FUNCTION_BLOCK Gebhardt_Speed
VAR_INPUT
	EN: BOOL;
	ModbusRTU: REFERENCE TO ModbusRTU;
	Address: BYTE := 101;
END_VAR
VAR_OUTPUT
	ENO: BOOL;
	Speed: LREAL;
END_VAR
VAR
	ModbusWord_T_Speed: ModbusReadWord;
END_VAR

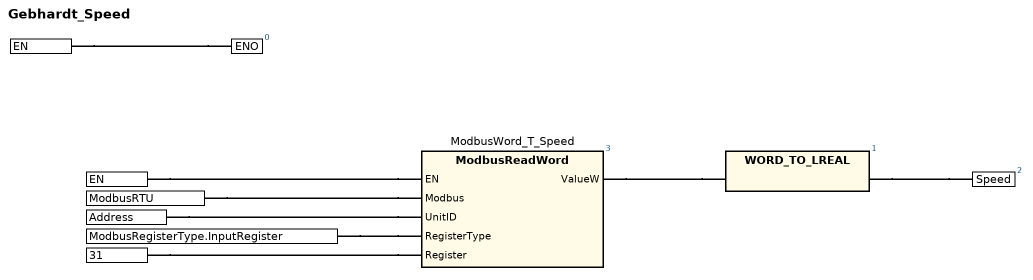
ENO := EN;
Speed := WORD_TO_LREAL(ModbusWord_T_Speed.ValueW);
ModbusWord_T_Speed(
    EN := EN,
    Modbus := ModbusRTU,
    UnitID := Address,
    RegisterType := ModbusRegisterType.InputRegister,
    Register := 31); // ModbusReadWord

END_FUNCTION_BLOCK

(* stored: Version 1.1.0.1, ProductVersion 3.1.4024.6
   POU Gebhardt_Speed: Id {00b88721-71e6-470f-a28b-f21d84461f04}, SpecialFunc None *)
